// TwinCAT 3 PLC project Project
// ProgramVersion: 3.1.4022.7
// libraries:
//   LCLS General, * (SLAC)
//   lcls-twincat-motion, * (SLAC)
//   Tc2_Standard, * (Beckhoff Automation GmbH)
//   Tc2_System, * (Beckhoff Automation GmbH)
//   Tc2_Utilities, * (Beckhoff Automation GmbH)
//   Tc3_EventLogger, * (Beckhoff Automation GmbH)
//   Tc3_Module, * (Beckhoff Automation GmbH)
// project tree:
//   GVLs/ DUT_Test.TcDUT, GVL.TcGVL
//   / PlcTask.TcTTO
//   POUs/ Main.TcPOU
// real-time tasks:
//   TASK PlcTask: cycle T#10ms, priority 20, ADS port 350
// motion (NC):
//   TASK NC-Task 1 SAF: cycle T#2ms, priority 4, ADS port 501
//   TASK NC-Task 1 SVB: cycle T#10ms, priority 8, ADS port 511
//   AXIS Axis 1 (id 1)
// variable links:
//   Project Instance <-> NC-Task 1 SAF/Axes/Axis 1
//     PlcTask Inputs/Main.M1.Axis.NcToPlc <-> Outputs/ToPlc
//     PlcTask Outputs/Main.M1.Axis.PlcToNc <-> Inputs/FromPlc

CONFIGURATION Project
    RESOURCE PLC ON TwinCAT3
        TASK PlcTask(INTERVAL := T#10ms, PRIORITY := 20);
        PROGRAM Main WITH PlcTask : Main;
    END_RESOURCE
END_CONFIGURATION

// ---- GVLs/DUT_Test.TcDUT
TYPE DUT_Test :
STRUCT

	{attribute 'pytmc' := '
		pv: intval
	'}
	intval : int;
	
END_STRUCT
END_TYPE

// ---- GVLs/GVL.TcGVL
{attribute 'qualified_only'}
VAR_GLOBAL
	CalculationEventClass: INT;
END_VAR

// ---- POUs/Main.TcPOU
PROGRAM Main
VAR
	{attribute 'pytmc' := '
    	pv: AXIS1
	'}
	M1: DUT_MotionStage;
	fbMotion1: FB_MotionStage;
	
	{attribute 'pytmc' := '
		pv: TEST:MAIN:SCALE
    	io: io
	'}
	scale : LREAL := 1.234;
	
	{attribute 'pytmc' := '
		pv: MY:DUT
		expand: :%.2d:
	'}
	test_arr : array[1..5] of DUT_Test;
	
	iLoop : UINT;
	
	{attribute 'pytmc' := '
		pv: TEST:LOGMESSAGE:
	'}
	fbLogger : FB_LogMessage;
	
	{attribute 'pytmc' := '
		pv: TEST:LOGHANDLER:
	'}
	fbLogHandler	: FB_LogHandler;
	
END_VAR

M1.bAllBackwardEnable := TRUE;
M1.bAllForwardEnable := TRUE;
M1.bBrakeRelease := TRUE;
M1.bPowerSelf := TRUE;
M1.nEnableMode := ENUM_StageEnableMode.STAGE_ENABLE_ALWAYS;

fbMotion1(stMotionStage:=M1);

iLoop := iLoop + 1;

if (iLoop MOD 100) = 0 then
	fbLogger.sJson := '{"user":"defined"}'; 
	fbLogger(sMsg:='the updated message', eSevr:=TcEventSeverity.Verbose, eSubsystem:= E_Subsystem.MOTION);
END_IF

fbLogHandler.fbLCLSListener.LogToVisualStudio := TRUE;
fbLogHandler();

END_PROGRAM
